// TIA Portal V19 export
VAR_GLOBAL   // PLC tag table "00_SAFETY_PEM_and_GEN"
   A01_PEm_Front AT %I1006.1 : Bool;   // 100DI1 - 142SB1,2,3,4,5,6 Emergency push buttons / 100DI1 - 142 E.Stop Area01 Front
   A01_PEm_Rear AT %I1006.2 : Bool;   // 100DI2 - 144SB1,2,3 Emergency push buttons / 100DI2 - 144 E.Stop Area01 Rear
   A02_PEm_Front AT %I1006.3 : Bool;   // 100DI3 - 146SB1,2,3,4 Emergency push buttons / 100DI3 - 146 E.Stop Area02 Front
   A02_PEm_Rear AT %I1013.0 : Bool;   // 101DI0 - 148SB1,2 Emergency push buttons / 101DI0 - 148 E.Stop Area02 Rear
   A03_PEm_Front_1 AT %I1200.0 : Bool;   // 200DI0 - 150SB1,2 Emergency push buttons / 200DI0 - 150 E.Stop Area03 Front 1
   A03_PEm_Rear_1 AT %I1300.0 : Bool;   // 250DI0 - 154SB1,2 Emergency push buttons / 300DI0 - 151 E.Stop Area03 Rear 2
   A01_Pb_SafetyReset AT %I102.0 : Bool;   // 158SH1 - MB1 safety reset button / 158SH1
   A01_Lp_SafetyReset AT %Q106.0 : Bool;   // 158SH1 - MB1 safety reset button lamp / 158SH1
   A02_Pb_SafetyReset AT %I102.1 : Bool;   // 158SH1 - MB1 safety reset button / 158SH2
   A02_Lp_SafetyReset AT %Q106.1 : Bool;   // 158SH1 - MB1 safety reset button / 158SH2
   A03_Pb_SafetyReset AT %I102.2 : Bool;   // 159SH1 - MB1 safety reset button / 159SH1
   A03_Lp_SafetyReset AT %Q106.2 : Bool;   // 159SH1 - MB1 safety reset button lamp / 159SH1
   A01_Sel_SetUp AT %I1013.1 : Bool;   // 101DI1 - 158SA1 Area 01 SetUp selector / 101DI1 - 158
   A02_Sel_SetUp AT %I1013.2 : Bool;   // 101DI2 - 158SA2 Area 02 SetUp selector / 101DI2 - 158
   A03_Sel_SetUp AT %I1013.3 : Bool;   // 101DI3 - 159SA1 Area 03 SetUp selector / 101DI3 - 159
   A03_PEm_Front_2 AT %I1400.0 : Bool;   // 300DI0 - 151SB1,2 Emergency push buttons / 350DI0 - 152 E.Stop Area03 Front 2
   A03_PEm_Rear_2 AT %I1400.1 : Bool;   // 300DI1 - 155SB1 Emergency push buttons / 250DI0 - 154 E.Stop Area03 Rear 2
   GEN_PEm AT %I1006.0 : Bool;   // 100DI0 - 140SB1,2,3,4,5 Emergency push buttons
   A03_PEm_Front_3 AT %I1500.0 : Bool;   // 350DI0 - 152SB1,2 Emergency push buttons / 350DI0 - 152 E.Stop Area03 Front 2
   A03_PEm_Rear_3 AT %I1500.1 : Bool;   // 350DI1 - 156SB1 Emergency push buttons / 250DI0 - 154 E.Stop Area03 Rear 2   {ExternalAccessible false}
   "495A2_NotUsed" AT %I1207.0 : Bool;
   "515A2_NotUsed" AT %I1307.0 : Bool;
END_VAR
